FUNCTION "FC_Dryer" : Void
{ S7_Optimized_Access := 'TRUE' }
VERSION : 1.0
// ==============================================================================
// FC_Sushka - Детальная диагностика (27 бит в DWORD)
// Fans: 0..6 (Breaker), 7..13 (FB)
// Burners: 14..15 (Breaker), 16..17 (FB), 18..19 (Temp), 20..21 (Alarm), 22..23 (Auto)
// Discharge: 24 (FB)
// Levels: 25 (High), 26 (Low)
// ==============================================================================
   VAR_INPUT
      Index : Int;
   END_VAR

   VAR_IN_OUT
      B : "UDT_BaseMechanism";
      D : "UDT_Dryer";
      R : "UDT_Dryer_Recipe";
   END_VAR

   VAR_TEMP
      i : Int;   // Итератор
      timeElapsed : Bool;
      elapsedMs : DInt;
      nowTck : DInt;
      anyFanFault : Bool;   // Флаг аварии любого вентилятора
      anyBurnerFault : Bool;   // Флаг аварии любой горелки
      stepTimeout : DInt;   // Задержка между шагами
      isLowLevelActive : Bool;   // Флаг срабатывания нижнего уровня
      isHighLevelActive : Bool;   // Флаг срабатывания верхнего уровня
      isStoppingFault : Bool;   // Флаг критической аварии (требующей останова сушилки)
      isBreakerFlt : Bool;
      isFbFlt : Bool;
      isTempFlt : Bool;
      isAlarmFlt : Bool;
      isAutoFlt : Bool;
      isFbWait : Bool;   // Флаг завершения задержки пуска для контроля фидбека
      tempWord : Word;
      m : DWord;   // Временная маска бита
      totalCycleMs : DInt;   // Общий цикл (Работа + Пауза)
      runTimeMs : DInt;   // Рассчитанное время включения
      scaledPower : Int;   // Для масштабирования AI_Power
      raw30Deg : DInt;   // 30 градусов в RAW (0-27648)
      rawTdNom : DInt;   // Рецептная температура сушки в RAW
      rawTpNom : DInt;   // Рецептная температура продукта в RAW
      rawTgNom : DInt;   // Рецептная температура газа в RAW
      rawPWNom : DInt;   // Рецептная температура PW в RAW
      avgTdRaw : DInt;   // Среднее значение датчиков 10..11 в RAW
      avgTpRaw : DInt;   // Значение датчика 14 в RAW
      avgTgRaw : DInt;   // Среднее значение датчиков 6..7 в RAW
      avgPWRaw : DInt;   // Значение датчика 15 в RAW
      rawHysDeg : DInt;   // Hysteresis в RAW
      isRecipeTempsReady : Bool;   // Все три рецептурные температуры достигнуты
      isRecipeTdOver : Bool;   // Перегрев Td
      isRecipeTpOver : Bool;   // Перегрев Tp
      isRecipeTgOver : Bool;   // Перегрев Tg
      isRecipePWOver : Bool;   // Перегрев PW
      isTempOver : Bool;   // Общий признак перегрева для блокировки горелок/выгрузки
      sensorSpan : DInt;   // Диапазон датчика (Max - Min)
      highLevelHoldMs : DInt;   // Время удержания уровня в мс
   END_VAR


BEGIN
	    #stepTimeout := 3000; // 3 секунды между включениями компонентов

	    // Расчет параметров масштабирования (оптимизировано)
	    #sensorSpan := INT_TO_DINT(#R.SensorMax - #R.SensorMin);
	    IF #sensorSpan <= 0 THEN
	        #sensorSpan := 700;
	    END_IF; // Защита от деления на 0

	    // Коэффициент пересчета Градус -> RAW
	    // (Value - Min) * 27648 / Span
	    #rawHysDeg := (#R.Hysteresis_Temp * 27648) / #sensorSpan;

	    #raw30Deg := (30 - INT_TO_DINT(#R.SensorMin)) * 27648 / #sensorSpan;
	    #rawTdNom := (INT_TO_DINT(#R.TdNom) - INT_TO_DINT(#R.SensorMin)) * 27648 / #sensorSpan;
	    #rawTpNom := (INT_TO_DINT(#R.TpNom) - INT_TO_DINT(#R.SensorMin)) * 27648 / #sensorSpan;
	    #rawTgNom := (INT_TO_DINT(#R.TgNom) - INT_TO_DINT(#R.SensorMin)) * 27648 / #sensorSpan;
	    #rawPWNom := (INT_TO_DINT(#R.PWNom) - INT_TO_DINT(#R.SensorMin)) * 27648 / #sensorSpan;

	    // Приводим время к миллисекундам один раз (предполагаем, что в рецепте СЕКУНДЫ)
	    #highLevelHoldMs := #R.Time_High_Level * 1000;

	    #avgTdRaw := (INT_TO_DINT(#D.Temps[10]) + INT_TO_DINT(#D.Temps[11])) / 2;
	    #avgTpRaw := INT_TO_DINT(#D.Temps[14]);
	    #avgTgRaw := (INT_TO_DINT(#D.Temps[6]) + INT_TO_DINT(#D.Temps[7])) / 2;
	    #avgPWRaw := INT_TO_DINT(#D.Temps[15]);
	    #isRecipeTempsReady := (#avgTdRaw >= #rawTdNom) AND (#avgTpRaw >= #rawTpNom) AND (#avgTgRaw >= #rawTgNom) AND (#avgPWRaw >= #rawPWNom);

	    // Логика гистерезиса: блокировка при перегреве +5, снятие при возврате к номиналу
	    // Td
	    IF (#avgTdRaw > (#rawTdNom + #rawHysDeg)) THEN
	        #isRecipeTdOver := TRUE;
	    ELSIF (#avgTdRaw <= #rawTdNom) THEN
	        #isRecipeTdOver := FALSE;
	    ELSE
	        #isRecipeTdOver := (#D.FLTCode AND DW#16#08000000) <> 0;
	    END_IF;
	    #isRecipeTdOver := #isRecipeTdOver AND ((#D.ForceCode AND DW#16#08000000) = 0);

	    // Tp
	    IF (#avgTpRaw > (#rawTpNom + #rawHysDeg)) THEN
	        #isRecipeTpOver := TRUE;
	    ELSIF (#avgTpRaw <= (#rawTpNom - #rawHysDeg)) THEN
	        #isRecipeTpOver := FALSE;
	    ELSE
	        #isRecipeTpOver := (#D.FLTCode AND DW#16#10000000) <> 0;
	    END_IF;
	    #isRecipeTpOver := #isRecipeTpOver AND ((#D.ForceCode AND DW#16#10000000) = 0);

	    // Tg
	    IF (#avgTgRaw > (#rawTgNom + #rawHysDeg)) THEN
	        #isRecipeTgOver := TRUE;
	    ELSIF (#avgTgRaw <= #rawTgNom) THEN
	        #isRecipeTgOver := FALSE;
	    ELSE
	        #isRecipeTgOver := (#D.FLTCode AND DW#16#20000000) <> 0;
	    END_IF;
	    #isRecipeTgOver := #isRecipeTgOver AND ((#D.ForceCode AND DW#16#20000000) = 0);

	    // PW
	    IF (#avgPWRaw > (#rawPWNom + #rawHysDeg)) THEN
	        #isRecipePWOver := TRUE;
	    ELSIF (#avgPWRaw <= #rawPWNom) THEN
	        #isRecipePWOver := FALSE;
	    ELSE
	        #isRecipePWOver := (#D.FLTCode AND DW#16#40000000) <> 0;
	    END_IF;
	    #isRecipePWOver := #isRecipePWOver AND ((#D.ForceCode AND DW#16#40000000) = 0);

	    #isTempOver := #isRecipeTdOver OR #isRecipeTpOver OR #isRecipeTgOver OR #isRecipePWOver;

	    // 1. Сброс аварий (RESET)
	    IF #B.Cmd = "CMD_RESET" THEN
	        #D.FLTCode := 16#0; // Сброс детальной маски
	        #B.FLTCode := 16#0; // Сброс базовой маски
	        IF #B.FLTCode = "FLT_NONE" AND #B.Status = "STS_FAULT" THEN
	            IF NOT #B.LocalManual THEN
	                #B.Status := "STS_IDLE";
	                #D.Status := "STS_IDLE";
	            ELSE
	                #B.Status := "STS_LOCAL";
	                #D.Status := "STS_IDLE";
	            END_IF;
	        END_IF;
	        IF #B.Enable_OK AND #B.Status = "STS_DISABLED" THEN
	            #B.Status := "STS_IDLE";
	            #D.Status := "STS_IDLE";
	        END_IF;
	    END_IF;

	    // 2. Мониторинг под-устройств (Вентиляторы и Горелки)
	    #anyFanFault := FALSE;
	    FOR #i := 0 TO 6 DO
	        #isBreakerFlt := NOT #D.Fans[#i].DI_Breaker_OK AND ((#D.ForceCode AND SHL(IN := DW#16#1, N := INT_TO_UINT(#i))) = 0);

	        #isFbWait := (#B.Status = "STS_RUNNING") OR (#B.Status = "STS_STARTING" AND #D.Step > (#i + 1));
	        #m := SHL(IN := DW#16#1, N := INT_TO_UINT(#i + 7)); // Бит 7..13 (Feedback)

	        // Контроль фидбека вентиляторов с задержкой 2с
	        IF #D.Fans[#i].DO_Run AND NOT #D.Fans[#i].DI_Feedback_OK AND #isFbWait AND ((#D.ForceCode AND #m) = 0) THEN
	            IF #D.FbTck[#i + 1] = 0 THEN
	                #D.FbTck[#i + 1] := TIME_TCK();
	                #isFbFlt := FALSE;
	            ELSE
	                #isFbFlt := "FC_TimeElapsedMs"(StartTck := #D.FbTck[#i + 1], TimeoutMs := 2000, ElapsedMs => #elapsedMs, NowTck => #nowTck);
	            END_IF;
	        ELSE
	            #D.FbTck[#i + 1] := 0;
	            #isFbFlt := FALSE;
	        END_IF;

	        IF #isBreakerFlt OR #isFbFlt THEN
	            #D.Fans[#i].Status := "STS_FAULT";
	            #anyFanFault := TRUE;
	            IF #isBreakerFlt THEN
	                #D.FLTCode := #D.FLTCode OR SHL(IN := DW#16#1, N := INT_TO_UINT(#i));
	            END_IF;
	            IF #isFbFlt THEN
	                #D.FLTCode := #D.FLTCode OR #m;
	            END_IF;
	        ELSIF NOT #D.Fans[#i].DO_Run THEN
	            IF #B.Status = "STS_STOPPING" AND #D.Step = (#i + 1) THEN
	                #D.Fans[#i].Status := "STS_STOPPING";
	            ELSE
	                #D.Fans[#i].Status := "STS_IDLE";
	            END_IF;
	        ELSE
	            IF #B.Status = "STS_STARTING" AND #D.Step = (#i + 1) THEN
	                #D.Fans[#i].Status := "STS_STARTING";
	            ELSE
	                #D.Fans[#i].Status := "STS_RUNNING";
	            END_IF;
	        END_IF;
	    END_FOR;

	    #anyBurnerFault := FALSE;
	    FOR #i := 0 TO 1 DO
	        #isBreakerFlt := NOT #D.Burners[#i].DI_Breaker_OK AND ((#D.ForceCode AND SHL(IN := DW#16#1, N := INT_TO_UINT(14 + #i))) = 0);
	        #isTempFlt := NOT #D.Burners[#i].DI_Temp_OK AND ((#D.ForceCode AND SHL(IN := DW#16#1, N := INT_TO_UINT(18 + #i))) = 0);
	        #isAlarmFlt := #D.Burners[#i].DI_Alarm AND ((#D.ForceCode AND SHL(IN := DW#16#1, N := INT_TO_UINT(20 + #i))) = 0);
	        #isAutoFlt := NOT #D.Burners[#i].DI_Auto_OK AND ((#D.ForceCode AND SHL(IN := DW#16#1, N := INT_TO_UINT(22 + #i))) = 0);

	        // Фидбек контролируется когда горелка включена и уже прошёл шаг её запуска
	        #isFbWait := #D.Burners[#i].DO_Run AND
	        (#B.Status = "STS_RUNNING" OR
	        (#B.Status = "STS_STARTING" AND #D.Step > (8 + #i)));

	        IF #D.Burners[#i].DO_Run AND (NOT #D.Burners[#i].DI_Feedback1_OK OR NOT #D.Burners[#i].DI_Feedback2_OK)
	            AND #isFbWait AND ((#D.ForceCode AND SHL(IN := DW#16#1, N := INT_TO_UINT(16 + #i))) = 0) THEN
	            IF #D.FbTck[#i + 8] = 0 THEN
	                #D.FbTck[#i + 8] := TIME_TCK();
	                #isFbFlt := FALSE;
	            ELSE
	                #isFbFlt := "FC_TimeElapsedMs"(StartTck := #D.FbTck[#i + 8], TimeoutMs := 2000, ElapsedMs => #elapsedMs, NowTck => #nowTck);
	            END_IF;
	        ELSE
	            #D.FbTck[#i + 8] := 0;
	            #isFbFlt := FALSE;
	        END_IF;

	        IF #isBreakerFlt OR #isTempFlt OR #isAlarmFlt OR #isFbFlt OR #isAutoFlt THEN
	            #D.Burners[#i].Status := "STS_FAULT";
	            #anyBurnerFault := TRUE;
	            IF #isBreakerFlt THEN
	                #D.FLTCode := #D.FLTCode OR SHL(IN := DW#16#1, N := INT_TO_UINT(14 + #i));
	            END_IF;
	            IF #isFbFlt THEN
	                #D.FLTCode := #D.FLTCode OR SHL(IN := DW#16#1, N := INT_TO_UINT(16 + #i));
	            END_IF;
	            IF #isTempFlt THEN
	                #D.FLTCode := #D.FLTCode OR SHL(IN := DW#16#1, N := INT_TO_UINT(18 + #i));
	            END_IF;
	            IF #isAlarmFlt THEN
	                #D.FLTCode := #D.FLTCode OR SHL(IN := DW#16#1, N := INT_TO_UINT(20 + #i));
	            END_IF;
	            IF #isAutoFlt THEN
	                #D.FLTCode := #D.FLTCode OR SHL(IN := DW#16#1, N := INT_TO_UINT(22 + #i));
	            END_IF;
	        ELSIF NOT #D.Burners[#i].DO_Run THEN
	            IF #B.Status = "STS_STOPPING" AND #D.Step = (8 + #i) THEN
	                #D.Burners[#i].Status := "STS_STOPPING";
	            ELSE
	                #D.Burners[#i].Status := "STS_IDLE";
	            END_IF;
	        ELSE
	            // DO_Run=TRUE:
	            // STARTING — шаг запуска этой горелки (Step = 8+i)
	            // RUNNING  — Step ушёл дальше (Step > 8+i)
	            IF #B.Status = "STS_STARTING" AND #D.Step = (8 + #i) THEN
	                #D.Burners[#i].Status := "STS_STARTING";
	            ELSE
	                #D.Burners[#i].Status := "STS_RUNNING";
	            END_IF;
	        END_IF;
	    END_FOR;

	    // 3. Выгрузка и Уровни
	    IF #D.Discharge.DO_Run AND NOT #D.Discharge.DI_Feedback_OK AND ((#D.ForceCode AND DW#16#1000000) = 0) THEN
	        IF #D.FbTck[10] = 0 THEN
	            #D.FbTck[10] := TIME_TCK();
	        ELSIF "FC_TimeElapsedMs"(StartTck := #D.FbTck[10], TimeoutMs := 2000, ElapsedMs => #elapsedMs, NowTck => #nowTck) THEN
	            #D.FLTCode := #D.FLTCode OR DW#16#1000000; // Бит 24
	        END_IF;
	    ELSE
	        #D.FbTck[10] := 0;
	    END_IF;

	    // Логика удержания верхнего уровня (Minimum Hold Time)
	    IF NOT #D.Levels.High_OK THEN
	        #D.FbTck[11] := TIME_TCK();
	    END_IF;

	    IF #D.FbTck[11] <> 0 THEN
	        #isHighLevelActive := TRUE;
	        // Удерживаем аварию до истечения времени И возврата датчика в норму
	        IF "FC_TimeElapsedMs"(StartTck := #D.FbTck[11], TimeoutMs := #highLevelHoldMs, ElapsedMs => #elapsedMs, NowTck => #nowTck) AND #D.Levels.High_OK THEN
	            #D.FbTck[11] := 0;
	            #isHighLevelActive := FALSE;
	        END_IF;
	    ELSE
	        #isHighLevelActive := FALSE;
	    END_IF;

	    // Очищуємо біти рівнів та перегрівів (25-30) перед перевіркою, щоб вони працювали динамічно
	    #D.FLTCode := #D.FLTCode AND DW#16#F9FFFFFF; // Сбрасываем только уровни (25,26), темп. контролируются логикой выше

	    IF #isHighLevelActive AND ((#D.ForceCode AND DW#16#2000000) = 0) THEN
	        #D.FLTCode := #D.FLTCode OR DW#16#2000000; // Бит 25
	    END_IF;
	    IF NOT #D.Levels.Low_OK AND ((#D.ForceCode AND DW#16#4000000) = 0) THEN
	        #D.FLTCode := #D.FLTCode OR DW#16#4000000; // Бит 26
	    END_IF;

	    // Устанавливаем или сбрасываем биты перегрева в маске согласно результатам гистерезиса
	    IF #isRecipeTdOver THEN
	        #D.FLTCode := #D.FLTCode OR DW#16#8000000;
	    ELSE
	        #D.FLTCode := #D.FLTCode AND NOT DW#16#8000000;
	    END_IF;

	    IF #isRecipeTpOver THEN
	        #D.FLTCode := #D.FLTCode OR DW#16#10000000;
	    ELSE
	        #D.FLTCode := #D.FLTCode AND NOT DW#16#10000000;
	    END_IF;

	    IF #isRecipeTgOver THEN
	        #D.FLTCode := #D.FLTCode OR DW#16#20000000;
	    ELSE
	        #D.FLTCode := #D.FLTCode AND NOT DW#16#20000000;
	    END_IF;

	    IF #isRecipePWOver THEN
	        #D.FLTCode := #D.FLTCode OR DW#16#40000000;
	    ELSE
	        #D.FLTCode := #D.FLTCode AND NOT DW#16#40000000;
	    END_IF;

	    #isLowLevelActive := (#D.FLTCode AND DW#16#4000000) <> 0;

	    // Критическая авария - любая кроме Верхнего/Нижнего уровней и Перегревов (25..30)
	    #isStoppingFault := (#D.FLTCode AND DW#16#81FFFFFF) <> 0;

	    // Связь с базовым механизмом: если есть реальная ошибка в S.FLTCode,
	    // ставим общую аварию в B.FLTCode для Арбитра и Маршрутов.
	    // Уровни (верхний/нижний) не должны давать глобальную аварийную зупинку.
	    IF (#D.FLTCode AND DW#16#F9FFFFFF) <> 0 THEN
	        #B.FLTCode := W#16#0001; // Просто "Авария" в базовом слоте
	    ELSE
	        #B.FLTCode := W#16#0000;
	    END_IF;

	    IF NOT #B.Enable_OK THEN
	        #B.Status := "STS_DISABLED";
	        #D.Step := 0;
	    ELSIF #B.LocalManual THEN
	        #B.Status := "STS_LOCAL";
	        #D.Step := 0;
	    ELSIF #isStoppingFault THEN // Останавливаем сушку только по критическим авариям
	        #B.Status := "STS_FAULT";
	        #D.Step := 0;
	    ELSE
	        CASE #B.Status OF
	            "STS_IDLE":
	                // Сушилка запускается ТОЛЬКО оператором вручную (OWNER_SCADA)
	                IF #B.Cmd = "CMD_START" AND #B.OwnerCur = "OWNER_SCADA" THEN
	                    // Сушилка готова к пуску если:
	                    // 1. Прошло время отдыха первого вентилятора
	                    // 2. Горелки в режиме AUTO
	                    #timeElapsed := #D.Fans[0].LastStopMs = 0 OR
	                    "FC_TimeElapsedMs"(StartTck := #D.Fans[0].LastStopMs,
	                                       TimeoutMs := 5000,
	                                       ElapsedMs => #elapsedMs,
	                                       NowTck => #nowTck);

	                    IF #timeElapsed AND #D.Burners[0].DI_Auto_OK AND #D.Burners[1].DI_Auto_OK THEN
	                        #B.Status := "STS_STARTING";
	                        #D.Step := 1;
	                        #D.StepStartTck := TIME_TCK();
	                    END_IF;
	                END_IF;

	            "STS_STARTING":
	                #timeElapsed := "FC_TimeElapsedMs"(StartTck := #D.StepStartTck,
	                                                   TimeoutMs := #stepTimeout,
	                                                   ElapsedMs => #elapsedMs,
	                                                   NowTck => #nowTck);
	                IF #timeElapsed THEN
	                    IF #D.Step < 9 THEN
	                        IF (#D.Step + 1) <= 7 THEN
	                            IF #D.Fans[#D.Step].LastStopMs = 0 OR "FC_TimeElapsedMs"(StartTck := #D.Fans[#D.Step].LastStopMs,
	                                                                                         TimeoutMs := 5000,
	                                                                                         ElapsedMs => #elapsedMs,
	                                                                                         NowTck => #nowTck) THEN
	                                #D.Step := #D.Step + 1;
	                                #D.StepStartTck := TIME_TCK();
	                            END_IF;
	                        ELSE
	                            #D.Step := #D.Step + 1;
	                            #D.StepStartTck := TIME_TCK();
	                        END_IF;
	                    ELSIF #D.Step = 9 THEN
	                        // Шаг 10: все компоненты запущены, переходим на ожидание температуры
	                        #D.Step := 10;
	                        #D.StepStartTck := TIME_TCK();
	                    ELSE
	                        // Шаг 10: ждём соответствия рецептурных температур
	                        IF #isRecipeTempsReady THEN
	                            IF #highLevelHoldMs <= 0 OR
	                                "FC_TimeElapsedMs"(StartTck := #D.StepStartTck,
	                                                   TimeoutMs := #highLevelHoldMs,
	                                                   ElapsedMs => #elapsedMs,
	                                                   NowTck => #nowTck) THEN
	                                #B.Status := "STS_RUNNING";
	                            END_IF;
	                        END_IF;
	                    END_IF;
	                END_IF;

	                IF #B.Cmd = "CMD_STOP" THEN
	                    #B.Status := "STS_STOPPING";
	                    #D.StepStartTck := TIME_TCK();
	                END_IF;

	            "STS_RUNNING":
	                // Авто-останов при пустой сушке и остывании до 30 градусов
	                IF #isLowLevelActive AND (INT_TO_DINT(#D.Temps[14]) < #raw30Deg) THEN
	                    #B.Status := "STS_STOPPING";
	                    #D.Step := 10;
	                    #D.StepStartTck := TIME_TCK();
	                END_IF;

	                IF #B.Cmd = "CMD_STOP" THEN
	                    #B.Status := "STS_STOPPING";
	                    #D.Step := 10; // Начинаем плавный останов с выключения горелок
	                    #D.StepStartTck := TIME_TCK();
	                END_IF;

	            "STS_STOPPING":
	                #timeElapsed := "FC_TimeElapsedMs"(StartTck := #D.StepStartTck,
	                                                   TimeoutMs := #stepTimeout,
	                                                   ElapsedMs => #elapsedMs,
	                                                   NowTck => #nowTck);
	                IF #timeElapsed THEN
	                    CASE #D.Step OF
	                        9, 10: // Постепенное выключение горелок
	                            #D.Step := #D.Step - 1;
	                            #D.StepStartTck := TIME_TCK();

	                        8: // Фаза охлаждения (Горелки уже OFF, Вентиляторы ON)
	                            IF (#avgTdRaw < #raw30Deg) AND (#avgTpRaw < #raw30Deg) AND
	                               (#avgTgRaw < #raw30Deg) AND (#avgPWRaw < #raw30Deg) THEN
	                                #D.Step := 7;
	                                #D.StepStartTck := TIME_TCK();
	                            END_IF;

	                        1..7: // Последовательное выключение вентиляторов
	                            // Защита от OMS: проверяем индекс перед записью
	                            IF #D.Step >= 1 AND #D.Step <= 7 THEN
	                                #D.Fans[#D.Step - 1].LastStopMs := TIME_TCK();
	                            END_IF;
	                            #D.Step := #D.Step - 1;
	                            #D.StepStartTck := TIME_TCK();

	                        0: // Завершение
	                            #B.Status := "STS_IDLE";
	                    END_CASE;
	                END_IF;
	        END_CASE;
	    END_IF;


	    // 5. Распределение команд на компоненты
	    IF #B.Status = "STS_FAULT" OR #B.Status = "STS_DISABLED" THEN
	        // Гасим всё при аварии или остановке
	        FOR #i := 0 TO 6 DO
	            #D.Fans[#i].DO_Run := FALSE;
	        END_FOR;
	        FOR #i := 0 TO 1 DO
	            #D.Burners[#i].DO_Run := FALSE;
	            #D.Burners[#i].AQ_Power := 0;
	        END_FOR;
	        #D.Discharge.DO_Run := FALSE;
	        #D.DischargeTimerTck := 0;
	    ELSE
	        // Управление вентиляторами (Шаги 1-7)
	        FOR #i := 0 TO 6 DO
	            IF #B.Status = "STS_RUNNING" THEN
	                #D.Fans[#i].DO_Run := TRUE;
	            ELSIF #B.Status = "STS_STARTING" AND #D.Step >= (#i + 1) THEN
	                #D.Fans[#i].DO_Run := TRUE;
	            ELSIF #B.Status = "STS_STOPPING" AND #D.Step >= (#i + 1) THEN
	                #D.Fans[#i].DO_Run := TRUE;
	            ELSE
	                #D.Fans[#i].DO_Run := FALSE;
	            END_IF;
	        END_FOR;

	        // Управление горелками (Шаги 8-9)
	        FOR #i := 0 TO 1 DO
	            #scaledPower := #D.Burners[#i].AI_Power;
	            IF #scaledPower < 0 THEN
	                #scaledPower := 0;
	            END_IF;
	            IF #scaledPower > 100 THEN
	                #scaledPower := 100;
	            END_IF;
	            #D.Burners[#i].AQ_Power := DINT_TO_INT((INT_TO_DINT(#scaledPower) * 27648) / 100);
	        END_FOR;

	        // Логика управления Горелкой 1 (Burner 1)
	        IF #isLowLevelActive THEN
	            #D.Burners[0].DO_Run := FALSE;
	            #D.Burners[0].AQ_Power := 0;
	        ELSIF (#B.Status = "STS_RUNNING" AND NOT #isTempOver) OR
	              (#B.Status = "STS_STARTING" AND #D.Step >= 8 AND NOT #isTempOver) OR
	              (#B.Status = "STS_STOPPING" AND #D.Step >= 9) THEN
	            #D.Burners[0].DO_Run := TRUE;
	        ELSE
	            #D.Burners[0].DO_Run := FALSE;
	            #D.Burners[0].AQ_Power := 0;
	        END_IF;

	        // Логика управления Горелкой 2 (Burner 2)
	        IF #isLowLevelActive THEN
	            #D.Burners[1].DO_Run := FALSE;
	            #D.Burners[1].AQ_Power := 0;
	        ELSIF (#B.Status = "STS_RUNNING" AND NOT #isTempOver) OR
	              (#B.Status = "STS_STARTING" AND #D.Step >= 9 AND NOT #isTempOver) OR
	              (#B.Status = "STS_STOPPING" AND #D.Step >= 10) THEN
	            #D.Burners[1].DO_Run := TRUE;
	        ELSE
	            #D.Burners[1].DO_Run := FALSE;
	            #D.Burners[1].AQ_Power := 0;
	        END_IF;

	        // Периодическое управление выгрузкой (PWM на базе процента)
	        IF #B.Status = "STS_RUNNING" AND #R.DischargePercent > 0 AND NOT #isLowLevelActive THEN
	            #runTimeMs := (INT_TO_DINT(#R.DischargePercent) * #R.MaxTimeRun) / 100;
	            #totalCycleMs := #runTimeMs + (INT_TO_DINT(#R.DischargePercent) * #R.MaxTimePause) / 100;

	            // Проверка прогресса текущего цикла
	            #timeElapsed := "FC_TimeElapsedMs"(StartTck := #D.DischargeTimerTck, TimeoutMs := #totalCycleMs, ElapsedMs => #elapsedMs, NowTck => #nowTck);

	            // Сброс или перезапуск таймера при завершении цикла
	            IF #D.DischargeTimerTck = 0 OR #timeElapsed THEN
	                #D.DischargeTimerTck := #nowTck;
	                #elapsedMs := 0;
	            END_IF;

	            #D.Discharge.DO_Run := #elapsedMs < #runTimeMs;
	        ELSE
	            #D.Discharge.DO_Run := FALSE;
	            #D.DischargeTimerTck := 0;
	        END_IF;
	    END_IF;

	    IF #B.Cmd <> "CMD_NONE" THEN
	        #B.LastCmd := #B.Cmd;
	    END_IF;
	    #B.Cmd := "CMD_NONE";
	    IF #D.ForceCode <> 0 THEN
	        #B.Force_Code := 1;
	    ELSE
	        #B.Force_Code := 0;
	    END_IF;

END_FUNCTION
